// TIA Portal project "4PUMPS_V16" (V16)
// Vorlageprojekt für das Buch mit Zielsystem S7-1200

(* hardware
DEVICE "S7-1200-Station_1"  S7-1200 Station
   slot 0: "Baugruppenträger_0"  Rack  V1.0
   slot 1: "PLC_1"  CPU 1211C DC/DC/DC  6ES7 211-1AE40-0XB0  V4.1
*)

// ===== PLC "PLC_1"  CPU 1211C DC/DC/DC =====

VAR_GLOBAL   // PLC tag table "Standard-Variablentabelle"
   "LL1" AT %I0.0 : Bool;
   "HL1" AT %I0.1 : Bool;
   "LL2" AT %I0.2 : Bool;
   "HL2" AT %I0.3 : Bool;
   "LL3" AT %I0.4 : Bool;
   "HL3" AT %I0.5 : Bool;
   "LL4" AT %I0.6 : Bool;
   "HL4" AT %I0.7 : Bool;
   "START" AT %I1.0 : Bool;
   "STOP" AT %I1.1 : Bool;
   "TANK 1 PUMP" AT %Q0.0 : Bool;
   "TANK 2 PUMP" AT %Q0.1 : Bool;
   "TANK 3 PUMP" AT %Q0.2 : Bool;
   "TANK 4 PUMP" AT %Q0.3 : Bool;
   "X" AT %M0.0 : Bool;
   "Y" AT %M0.1 : Bool;
END_VAR

FUNCTION "MHJ-PLC-Lab-Function-S71200" : Void   // FC9000, SCL
{ S7_Optimized_Access := 'TRUE' }
VERSION : 0.1
   VAR_TEMP
      rdTimeReturn : Int;
      outputTime : DTL;
      SyncVal : Byte;
      forVal : Int;
      forVal_2 : Int;
      Value : Byte;
   END_VAR
   VAR CONSTANT
      CompVal : Byte := 16#34;
      Value_01 : Byte := 16#11;
      Value_01_DW : DWord := 16#A165_D992;
      Value_02_DW : DWord := 16#58BE_4401;
   END_VAR
BEGIN

   #Value:=PEEK(area := 16#82,
        dbNumber := 0,
        byteOffset := 511);
   #Value := #Value + 1;

   POKE(area := 16#82,
        dbNumber := 0,
        byteOffset := 511,
        value := #Value);

   POKE(area:=16#81,
        dbNumber:=0,
        byteOffset:=1016,
        value:=#Value_01_DW);
   POKE(area := 16#81,
        dbNumber := 0,
        byteOffset := 1020,
        value := #Value_02_DW);

   POKE(area := 16#81,
        dbNumber := 0,
        byteOffset := 511,
        value := B#16#00);

   FOR #forVal := 0 TO 120 DO
       FOR #forVal_2:=0 TO 10 DO
           #rdTimeReturn:=RD_SYS_T(#outputTime);
           #rdTimeReturn := WR_SYS_T(#outputTime);
           #rdTimeReturn := RD_SYS_T(#outputTime);
           #rdTimeReturn := WR_SYS_T(#outputTime);
       END_FOR;
       #SyncVal:= PEEK(area := 16#81,
                      dbNumber := 0,
                      byteOffset := 511);
       IF #SyncVal = #CompVal THEN
          GOTO M_1;
       END_IF;
   END_FOR;
   RETURN;

   M_1:
   POKE(area := 16#81,
        dbNumber := 0,
        byteOffset := 511,
        value := B#16#0);
END_FUNCTION

ORGANIZATION_BLOCK "Main"   // OB1, LAD, ProgramCycle
TITLE = "Main Program Sweep (Cycle)"
{ S7_Optimized_Access := 'TRUE' }
VERSION : 0.1
   VAR_INPUT
      Initial_Call : Bool;   // Initial call of this OB
      Remanence : Bool;   // =True, if remanent data are available
   END_VAR
BEGIN

REGION Network 1: Konnektierungsbaustein für PLC-Lab
   // Im Netzwerk 1 wird der Konnektierungsbaustein für PLC-Lab aufgerufen.
   // Dieser Aufruf darf nicht entfernt werden!
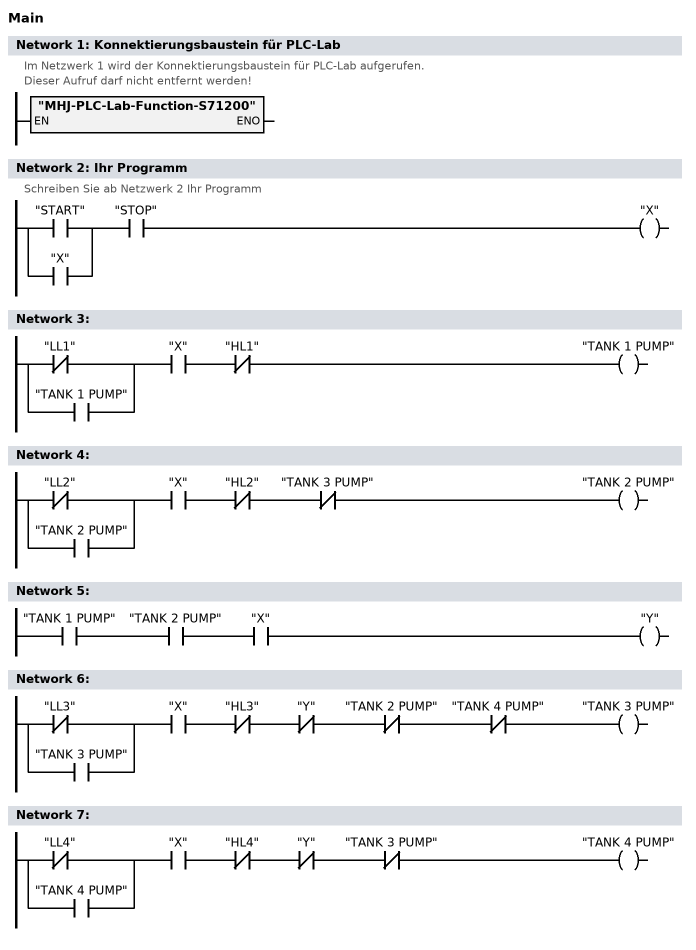
   RUNG wire#powerrail
      "MHJ-PLC-Lab-Function-S71200"()
   END_RUNG
   // the same network as SCL:
   "MHJ-PLC-Lab-Function-S71200"();
END_REGION

REGION Network 2: Ihr Programm
   // Schreiben Sie ab Netzwerk 2 Ihr Programm
   RUNG wire#powerrail
      Contact( "START" )
      wire#w1
      Contact( "STOP" )
      Coil( "X" )
   END_RUNG
   RUNG wire#powerrail
      Contact( "X" )
   END_RUNG wire#w1
   // the same network as SCL:
   "X" := ("START" OR "X") AND "STOP";
END_REGION

REGION Network 3
   RUNG wire#powerrail
      I_Contact( "LL1" )
      wire#w1
      Contact( "X" )
      I_Contact( "HL1" )
      Coil( "TANK 1 PUMP" )
   END_RUNG
   RUNG wire#powerrail
      Contact( "TANK 1 PUMP" )
   END_RUNG wire#w1
   // the same network as SCL:
   "TANK 1 PUMP" := (NOT "LL1" OR "TANK 1 PUMP") AND "X" AND NOT "HL1";
END_REGION

REGION Network 4
   RUNG wire#powerrail
      I_Contact( "LL2" )
      wire#w1
      Contact( "X" )
      I_Contact( "HL2" )
      I_Contact( "TANK 3 PUMP" )
      Coil( "TANK 2 PUMP" )
   END_RUNG
   RUNG wire#powerrail
      Contact( "TANK 2 PUMP" )
   END_RUNG wire#w1
   // the same network as SCL:
   "TANK 2 PUMP" := (NOT "LL2" OR "TANK 2 PUMP") AND "X" AND NOT "HL2" AND NOT "TANK 3 PUMP";
END_REGION

REGION Network 5
   RUNG wire#powerrail
      Contact( "TANK 1 PUMP" )
      Contact( "TANK 2 PUMP" )
      Contact( "X" )
      Coil( "Y" )
   END_RUNG
   // the same network as SCL:
   "Y" := "TANK 1 PUMP" AND "TANK 2 PUMP" AND "X";
END_REGION

REGION Network 6
   RUNG wire#powerrail
      I_Contact( "LL3" )
      wire#w1
      Contact( "X" )
      I_Contact( "HL3" )
      I_Contact( "Y" )
      I_Contact( "TANK 2 PUMP" )
      I_Contact( "TANK 4 PUMP" )
      Coil( "TANK 3 PUMP" )
   END_RUNG
   RUNG wire#powerrail
      Contact( "TANK 3 PUMP" )
   END_RUNG wire#w1
   // the same network as SCL:
   "TANK 3 PUMP" := (NOT "LL3" OR "TANK 3 PUMP") AND "X" AND NOT "HL3" AND NOT "Y" AND NOT "TANK 2 PUMP" AND NOT "TANK 4 PUMP";
END_REGION

REGION Network 7
   RUNG wire#powerrail
      I_Contact( "LL4" )
      wire#w1
      Contact( "X" )
      I_Contact( "HL4" )
      I_Contact( "Y" )
      I_Contact( "TANK 3 PUMP" )
      Coil( "TANK 4 PUMP" )
   END_RUNG
   RUNG wire#powerrail
      Contact( "TANK 4 PUMP" )
   END_RUNG wire#w1
   // the same network as SCL:
   "TANK 4 PUMP" := (NOT "LL4" OR "TANK 4 PUMP") AND "X" AND NOT "HL4" AND NOT "Y" AND NOT "TANK 3 PUMP";
END_REGION
END_ORGANIZATION_BLOCK